# EPICS autosave request: iocBoot/ioc1/dbSave/23i_MO_Ps_.req
%
% BURT Request File
%
% 23i:MO:Ps:  Monochromator Positioning (alignment)
%

file $(DIR)/assy.req ASSY=23i:MO:Ps
file $(DIR)/mtr1.req MTR1=23i:MO:mz
file $(DIR)/mtr1.req MTR1=23i:MO:my
file $(DIR)/drv1.req DRV1=23i:MO:Z
file $(DIR)/drv1.req DRV1=23i:MO:Y
